{attribute 'TcGenerated'}
// This function has been automatically generated from the project information.
VAR_GLOBAL CONSTANT
	{attribute 'const_non_replaced'}
	{attribute 'linkalways'}
	stLibVersion_ProfilerLib : ST_LibVersion := (iMajor := 0, iMinor := 0, iBuild := 0, iRevision := 1, sVersion := '0.0.0.1');
END_VAR

(* stored: Version 1.1.0.1, ProductVersion 3.1.4020.12
   GVL Global_Version: Id {c1e46cc5-befe-4132-944c-b0734b2499a3} *)
